KUKA KRL program: masref_user.src, masref_user.dat

--- masref_user.src ---
&ACCESS RVO1
&REL 1
&COMMENT Mastering Reference User Program
&PARAM DISKPATH = KRC:\R1\Program
DEF MasRef_USER()
END

GLOBAL DEF MASREFSTARTG1()
;FOLD Teach path and position for reference group 1
;ENDFOLD

END

GLOBAL DEF MASREFBACKG1()
;FOLD Teach path back for reference group 1
;ENDFOLD

END

GLOBAL DEF MASREFSTARTG2()
;FOLD Teach path and position for reference group 2
;ENDFOLD

END

GLOBAL DEF MASREFBACKG2()
;FOLD Teach path back for reference group 2
;ENDFOLD

END

GLOBAL DEF MASREFSTARTG3()
;FOLD Teach path and position for reference group 3
;ENDFOLD

END

GLOBAL DEF MASREFBACKG3()
;FOLD Teach path back for reference group 3
;ENDFOLD

END

--- masref_user.dat ---
&ACCESS RVO1
DEFDAT MasRef_User
;FOLD EXTERNAL DECLARATIONS;%{PE}%MKUKATPBASIS,%CEXT,%VCOMMON,%P
;FOLD GRIPPERTECH EXT
  EXT  H50 (INT:IN, INT:IN ,INT:IN ,GRP_TYP:IN)
;ENDFOLD (GRIPPERTECH EXT)
;FOLD SPOTTECH EXT
  EXT  USERSPOT (S_COMMAND  :IN, SPOT_TYPE:IN)
;ENDFOLD (SPOTTECH EXT)
;FOLD BASISTECH EXT;%{PE}%MKUKATPBASIS,%CEXT,%VEXT,%P
  EXT  BAS (BAS_COMMAND  :IN,REAL  :IN )
;ENDFOLD (BASISTECH EXT)
;FOLD USER EXT;%{E}%MKUKATPUSER,%CEXT,%VEXT,%P
;Make here your modifications

;ENDFOLD (USER EXT)
;ENDFOLD (EXTERNAL DECLERATIONS)
ENDDAT
